// Mitsubishi GX Works2 project: VentiladoresV5   PLC: FX3G
// VentiladoresAndreDC

// global labels: Global1
VAR_GLOBAL
  Frecuencia_Actual_Cocina_Boilers AT D100 : INT;
  Corriente_Actual_Cocina_Boilers AT D102 : INT;
  Alarma_Cocina_Boilers AT M0 : BOOL;
  Automatico_Cocina_Boilers AT M1 : BOOL;
  Encender_Manual_Cocina_Boilers AT M2 : BOOL;
  Apagar_Manual_Cocina_Boilers AT M3 : BOOL;
  Reset_Alarma_Cocina_Boilers AT M4 : BOOL;
  Hora_Encendido_Cocina_Boilers AT D104 : INT;
  Minuto_Encendido_Cocina_Boilers AT D106 : INT;
  Hora_Apagado_Cocina_Boilers AT D108 : INT;
  Minuto_Apagado_Cocina_Boilers AT D110 : INT;
  SP_Velocidad_Cocina_Boilers AT D112 : INT;
  Alarma_Suministro1 AT M10 : BOOL;
  Automatico_Suministro1 AT M11 : BOOL;
  Encender_Manual_Suministro1 AT M12 : BOOL;
  Apagar_Manual_Suministro1 AT M13 : BOOL;
  Reset_Alarma_Suministro1 AT M14 : BOOL;
  Frecuencia_Actual_Suministro1 AT D114 : INT;
  Corriente_Actual_Suministro1 AT D116 : INT;
  Hora_Encendido_Suministro1 AT D118 : INT;
  Minuto_Encendido_Suministro1 AT D120 : INT;
  Hora_Apagado_Suministro1 AT D122 : INT;
  Minuto_Apagado_Suministro1 AT D124 : INT;
  SP_Velocidad_Suministro1 AT D126 : INT;
  Alarma_Suministro2 AT M20 : BOOL;
  Automatico_Suministro2 AT M21 : BOOL;
  Encender_Manual_Suministro2 AT M22 : BOOL;
  Apagar_Manual_Suministro2 AT M23 : BOOL;
  Reset_Alarma_Suministro2 AT M24 : BOOL;
  Frecuencia_Actual_Suministro2 AT D128 : INT;
  Corriente_Actual_Suministro2 AT D130 : INT;
  Hora_Encendido_Suministro2 AT D132 : INT;
  Minuto_Encendido_Suministro2 AT D134 : INT;
  Hora_Apagado_Suministro2 AT D136 : INT;
  Minuto_Apagado_Suministro2 AT D138 : INT;
  SP_Velocidad_Suministro2 AT D140 : INT;
  Alarma_Cocina_Fria AT M30 : BOOL;
  Automatico_Cocina_Fria AT M31 : BOOL;
  Encender_Manual_Cocina_Fria AT M32 : BOOL;
  Apagar_Manual_Cocina_Fria AT M33 : BOOL;
  Reset_Alarma_Cocina_Fria AT M34 : BOOL;
  Frecuencia_Actual_Cocina_Fria AT D142 : INT;
  Corriente_Actual_Cocina_Fria AT D144 : INT;
  Hora_Encendido_Cocina_Fria AT D146 : INT;
  Minuto_Encendido_Cocina_Fria AT D148 : INT;
  Hora_Apagado_Cocina_Fria AT D150 : INT;
  Minuto_Apagado_Cocina_Fria AT D152 : INT;
  SP_Velocidad_Cocina_Fria AT D154 : INT;
  Alarma_Campana_Grande AT M40 : BOOL;
  Automatico_Campana_Grande AT M41 : BOOL;
  Encender_Manual_Campana_Grande AT M42 : BOOL;
  Apagar_Manual_Campana_Grande AT M43 : BOOL;
  Reset_Alarma_Campana_Grande AT M44 : BOOL;
  Frecuencia_Actual_Campana_Grande AT D156 : INT;
  Corriente_Actual_Campana_Grande AT D158 : INT;
  Hora_Encendido_Campana_Grande AT D160 : INT;
  Minuto_Encendido_Campana_Grande AT D162 : INT;
  Hora_Apagado_Campana_Grande AT D164 : INT;
  Minuto_Apagado_Campana_Grande AT D166 : INT;
  SP_Velocidad_Campana_Grande AT D168 : INT;
  Alarma_Fachada1 AT M50 : BOOL;
  Automatico_Fachada1 AT M51 : BOOL;
  Encender_Manual_Fachada1 AT M52 : BOOL;
  Apagar_Manual_Fachada1 AT M53 : BOOL;
  Reset_Alarma_Fachada1 AT M54 : BOOL;
  Frecuencia_Actual_Fachada1 AT D170 : INT;
  Corriente_Actual_Fachada1 AT D172 : INT;
  Hora_Encendido_Fachada1 AT D174 : INT;
  Minuto_Encendido_Fachada1 AT D176 : INT;
  Hora_Apagado_Fachada1 AT D178 : INT;
  Minuto_Apagado_Fachada1 AT D180 : INT;
  SP_Velocidad_Fachada1 AT D182 : INT;
  Alarma_Fachada2 AT M60 : BOOL;
  Automatico_Fachada2 AT M61 : BOOL;
  Encender_Manual_Fachada2 AT M62 : BOOL;
  Apagar_Manual_Fachada2 AT M63 : BOOL;
  Reset_Alarma_Fachada2 AT M64 : BOOL;
  Frecuencia_Actual_Fachada2 AT D184 : INT;
  Corriente_Actual_Fachada2 AT D186 : INT;
  Hora_Encendido_Fachada2 AT D188 : INT;
  Minuto_Encendido_Fachada2 AT D190 : INT;
  Hora_Apagado_Fachada2 AT D192 : INT;
  Minuto_Apagado_Fachada2 AT D194 : INT;
  SP_Velocidad_Fachada2 AT D196 : INT;
  Alarma_Cocina_Terraza AT M70 : BOOL;
  Automatico_Cocina_Terraza AT M71 : BOOL;
  Encender_Manual_Cocina_Terraza AT M72 : BOOL;
  Apagar_Manual_Cocina_Terraza AT M73 : BOOL;
  Reset_Alarma_Cocina_Terraza AT M74 : BOOL;
  Frecuencia_Actual_Cocina_Terraza AT D198 : INT;
  Corriente_Actual_Cocina_Terraza AT D200 : INT;
  Hora_Encendido_Cocina_Terraza AT D202 : INT;
  Minuto_Encendido_Cocina_Terraza AT D204 : INT;
  Hora_Apagado_Cocina_Terraza AT D206 : INT;
  Minuto_Apagado_Cocina_Terraza AT D208 : INT;
  SP_Velocidad_Cocina_Terraza AT D210 : INT;
  Cambiar_SP_Cocina_Boilers AT M5 : BOOL;
  Cambiar_SP_Suministro1 AT M15 : BOOL;
  Cambiar_SP_Suminsitro2 AT M25 : BOOL;
  Cambiar_SP_Cocina_Fria AT M35 : BOOL;
  Cambiar_SP_Campana_Grande AT M45 : BOOL;
  Cambiar_SP_Fachada1 AT M55 : BOOL;
  Cambiar_SP_Fachada2 AT M65 : BOOL;
  Cambiar_SP_Terraza AT M75 : BOOL;
  Ultima_Alarma_Cocina_Boilers AT D212 : INT;
  Ultima_Alarma_Suministro1 AT D214 : INT;
  Ultima_Alarma_Suministro2 AT D216 : INT;
  Ultima_Alarma_Cocina_Fria AT D218 : INT;
  Ultima_Alarma_Campana_Grande AT D220 : INT;
  Ultima_Alarma_Fachada1 AT D222 : INT;
  Ultima_Alarma_Fachada2 AT D224 : INT;
  Ultima_Alarma_Cocina_Terraza AT D226 : INT;
END_VAR

// task Task_01 (event TRUE, interval 0, priority 31): Inicio_Modbus, Campana_Grande, Cocina_Boilers, Cocina_Fria, Cocina_Terraza, Fachada1, Fachada2, Suministro1, Suministro2

PROGRAM Inicio_Modbus
(* structured ladder/FBD written out as ST: instructions are called as NAME(EN, inputs, outputs); _pN, _eN, _tN stand for wires *)
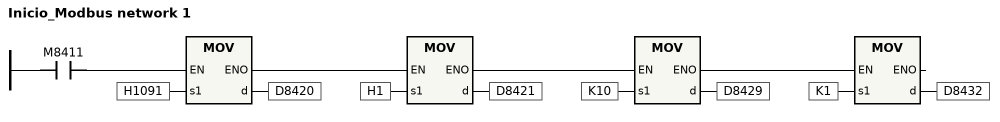
(* network 1 *)
_e1 := MOV(M8411, H1091, D8420);
_e2 := MOV(_e1, H1, D8421);
_e3 := MOV(_e2, K10, D8429);
MOV(_e3, K1, D8432);
END_PROGRAM

FUNCTION_BLOCK Comparador_Horario
VAR_INPUT
  Minuto_Encendido : INT;
  Hora_Encendido : INT;
  Minuto_Apagado : INT;
  Hora_Apagado : INT;
END_VAR
VAR
  Minuto_Encendido_Ok : BOOL;
  Hora_Encendido_Ok : BOOL;
  Minuto_Apagado_Ok : BOOL;
  Hora_Apagado_Ok : BOOL;
END_VAR
VAR_OUTPUT
  Dentro_Horario : BOOL;
END_VAR
VAR
  Encender : BOOL;
  Apagar : BOOL;
END_VAR
(* structured ladder/FBD written out as ST: instructions are called as NAME(EN, inputs, outputs); _pN, _eN, _tN stand for wires *)
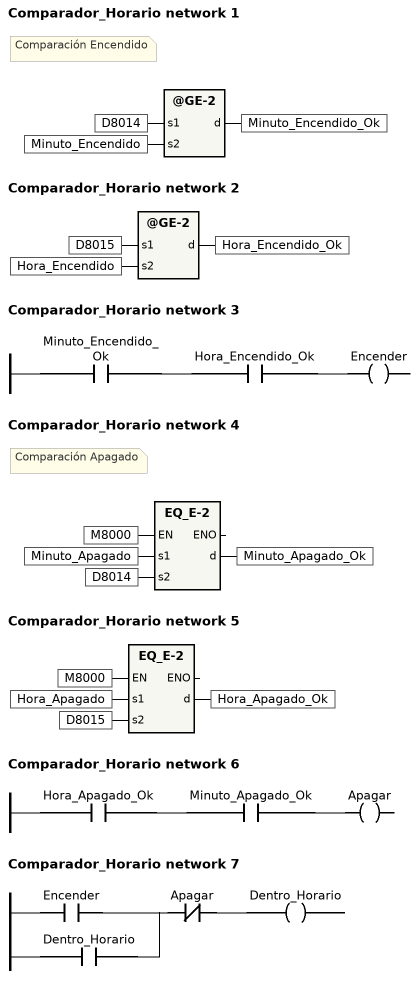
(* network 1 *)
(* Comparación Encendido *)
Minuto_Encendido_Ok := @GE-2(D8014, Minuto_Encendido);
(* network 2 *)
Hora_Encendido_Ok := @GE-2(D8015, Hora_Encendido);
(* network 3 *)
Encender := Minuto_Encendido_Ok AND Hora_Encendido_Ok;
(* network 4 *)
(* Comparación Apagado *)
EQ_E(M8000, Minuto_Apagado, D8014, Minuto_Apagado_Ok);
(* network 5 *)
EQ_E(M8000, Hora_Apagado, D8015, Hora_Apagado_Ok);
(* network 6 *)
Apagar := Hora_Apagado_Ok AND Minuto_Apagado_Ok;
(* network 7 *)
Dentro_Horario := (Encender OR Dentro_Horario) AND NOT Apagar;
END_FUNCTION_BLOCK

FUNCTION_BLOCK Control_Variador_Mitsubishi
VAR_INPUT
  Automatico : BOOL;
  Encender_Manual : BOOL;
  Hora_Encendido : INT;
  Minuto_Encendido : INT;
  SP_Velocidad : INT;
  Direccion_Modbus : INT;
END_VAR
VAR
  Comparador_Horario_1 : Comparador_Horario;
END_VAR
VAR_INPUT
  Minuto_Apagado : INT;
  Hora_Apagado : INT;
END_VAR
VAR
  Horario_Ok : BOOL;
  Encender_Variador_Automatico : BOOL;
  Apagar_Variador_Automatico : BOOL;
END_VAR
VAR_INPUT
  Apagar_Manual : BOOL;
END_VAR
VAR
  TP_1 : TP;
  TP_2 : TP;
END_VAR
VAR_INPUT
  Reset_Alarma : BOOL;
  Cambiar_SP : BOOL;
END_VAR
(* structured ladder/FBD written out as ST: instructions are called as NAME(EN, inputs, outputs); _pN, _eN, _tN stand for wires *)
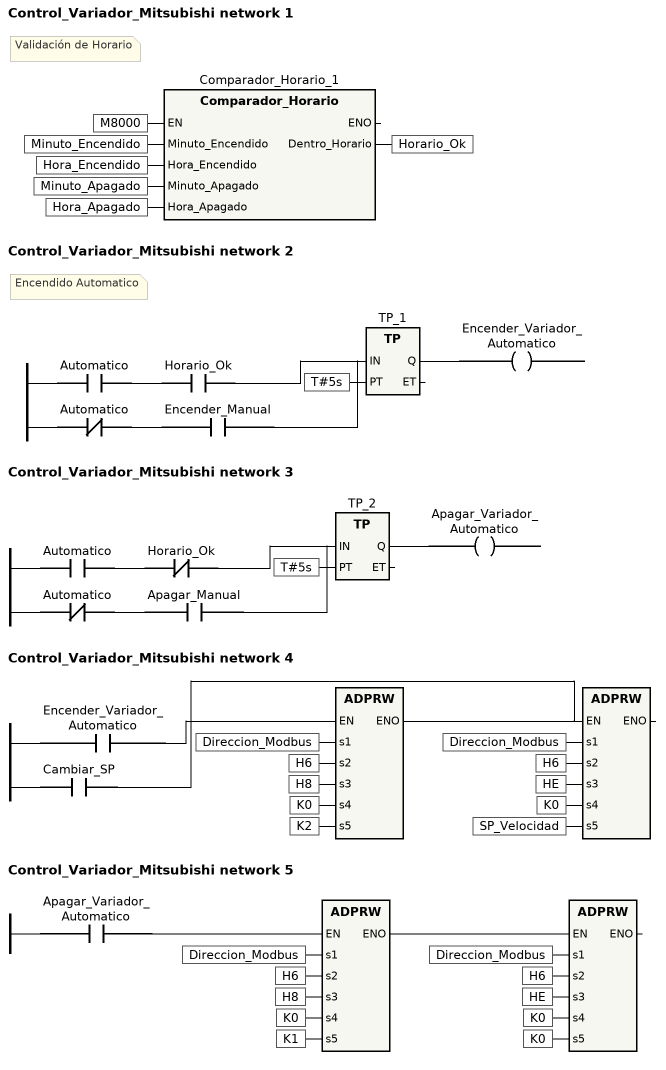
(* network 1 *)
(* Validación de Horario *)
Comparador_Horario_1(EN := M8000, Minuto_Encendido := Minuto_Encendido, Hora_Encendido := Hora_Encendido, Minuto_Apagado := Minuto_Apagado, Hora_Apagado := Hora_Apagado, Dentro_Horario => Horario_Ok);
(* network 2 *)
(* Encendido Automatico *)
TP_1(IN := (Automatico AND Horario_Ok) OR (NOT Automatico AND Encender_Manual), PT := T#5s);
Encender_Variador_Automatico := TP_1.Q;
(* network 3 *)
TP_2(IN := (Automatico AND NOT Horario_Ok) OR (NOT Automatico AND Apagar_Manual), PT := T#5s);
Apagar_Variador_Automatico := TP_2.Q;
(* network 4 *)
_e1 := ADPRW(Encender_Variador_Automatico, Direccion_Modbus, H6, H8, K0, K2);
ADPRW(_e1 OR Cambiar_SP, Direccion_Modbus, H6, HE, K0, SP_Velocidad);
(* network 5 *)
_e1 := ADPRW(Apagar_Variador_Automatico, Direccion_Modbus, H6, H8, K0, K1);
ADPRW(_e1, Direccion_Modbus, H6, HE, K0, K0);
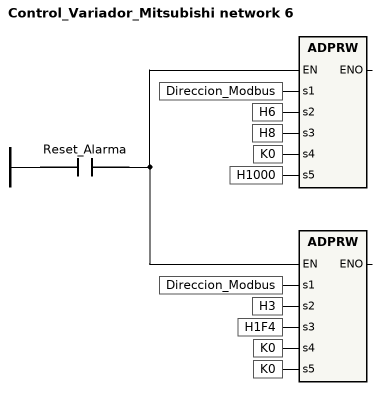
(* network 6 *)
ADPRW(Reset_Alarma, Direccion_Modbus, H6, H8, K0, H1000);
ADPRW(Reset_Alarma, Direccion_Modbus, H3, H1F4, K0, K0);
END_FUNCTION_BLOCK

FUNCTION_BLOCK Lectura_Variador_Mitsubishi
VAR_INPUT
  Direccion_Modbus : INT;
END_VAR
VAR_OUTPUT
  Frecuencia_Actual : INT;
  Corriente_Actual : INT;
  Alarma : BOOL;
END_VAR
VAR
  Estado_VFD : INT;
END_VAR
VAR_OUTPUT
  Ultima_Alarma : INT;
END_VAR
(* structured ladder/FBD written out as ST: instructions are called as NAME(EN, inputs, outputs); _pN, _eN, _tN stand for wires *)
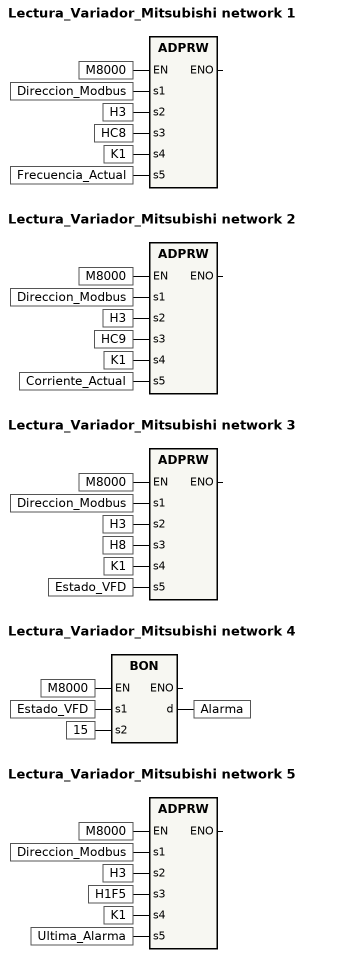
(* network 1 *)
ADPRW(M8000, Direccion_Modbus, H3, HC8, K1, Frecuencia_Actual);
(* network 2 *)
ADPRW(M8000, Direccion_Modbus, H3, HC9, K1, Corriente_Actual);
(* network 3 *)
ADPRW(M8000, Direccion_Modbus, H3, H8, K1, Estado_VFD);
(* network 4 *)
BON(M8000, Estado_VFD, 15, Alarma);
(* network 5 *)
ADPRW(M8000, Direccion_Modbus, H3, H1F5, K1, Ultima_Alarma);
END_FUNCTION_BLOCK

PROGRAM Cocina_Boilers
VAR
  Lectura_Variador_Mitsubishi_1 : Lectura_Variador_Mitsubishi;
  Control_Variador_Mitsubishi_1 : Control_Variador_Mitsubishi;
END_VAR
(* structured ladder/FBD written out as ST: instructions are called as NAME(EN, inputs, outputs); _pN, _eN, _tN stand for wires *)
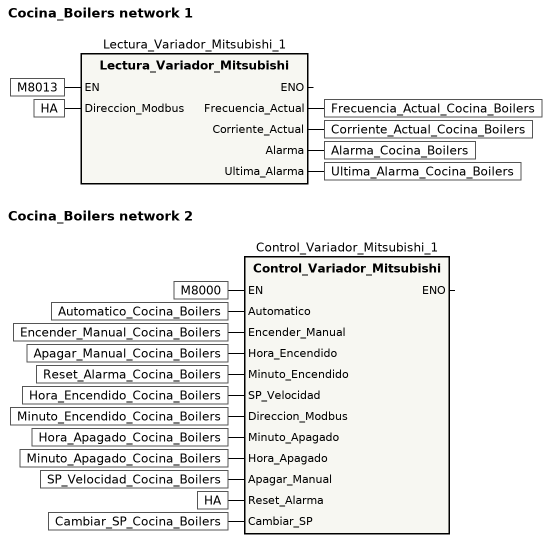
(* network 1 *)
Lectura_Variador_Mitsubishi_1(EN := M8013, Direccion_Modbus := HA, Frecuencia_Actual => Frecuencia_Actual_Cocina_Boilers, Corriente_Actual => Corriente_Actual_Cocina_Boilers, Alarma => Alarma_Cocina_Boilers, Ultima_Alarma => Ultima_Alarma_Cocina_Boilers);
(* network 2 *)
Control_Variador_Mitsubishi_1(EN := M8000, Automatico := Automatico_Cocina_Boilers, Encender_Manual := Encender_Manual_Cocina_Boilers, Hora_Encendido := Apagar_Manual_Cocina_Boilers, Minuto_Encendido := Reset_Alarma_Cocina_Boilers, SP_Velocidad := Hora_Encendido_Cocina_Boilers, Direccion_Modbus := Minuto_Encendido_Cocina_Boilers, Minuto_Apagado := Hora_Apagado_Cocina_Boilers, Hora_Apagado := Minuto_Apagado_Cocina_Boilers, Apagar_Manual := SP_Velocidad_Cocina_Boilers, Reset_Alarma := HA, Cambiar_SP := Cambiar_SP_Cocina_Boilers);
END_PROGRAM

FUNCTION_BLOCK Control_Variador_Altivar
VAR_INPUT
  Automatico : BOOL;
  Encender_Manual : BOOL;
  Hora_Encendido : INT;
  Minuto_Encendido : INT;
  SP_Velocidad : INT;
  Direccion_Modbus : INT;
END_VAR
VAR
  Comparador_Horario_1 : Comparador_Horario;
END_VAR
VAR_INPUT
  Minuto_Apagado : INT;
  Hora_Apagado : INT;
END_VAR
VAR
  Horario_Ok : BOOL;
  Encender_Variador_Automatico : BOOL;
  Apagar_Variador_Automatico : BOOL;
END_VAR
VAR_INPUT
  Apagar_Manual : BOOL;
END_VAR
VAR
  TP_1 : TP;
  TP_2 : TP;
END_VAR
VAR_INPUT
  Reset_Alarma : BOOL;
  Cambiar_SP : BOOL;
END_VAR
(* structured ladder/FBD written out as ST: instructions are called as NAME(EN, inputs, outputs); _pN, _eN, _tN stand for wires *)
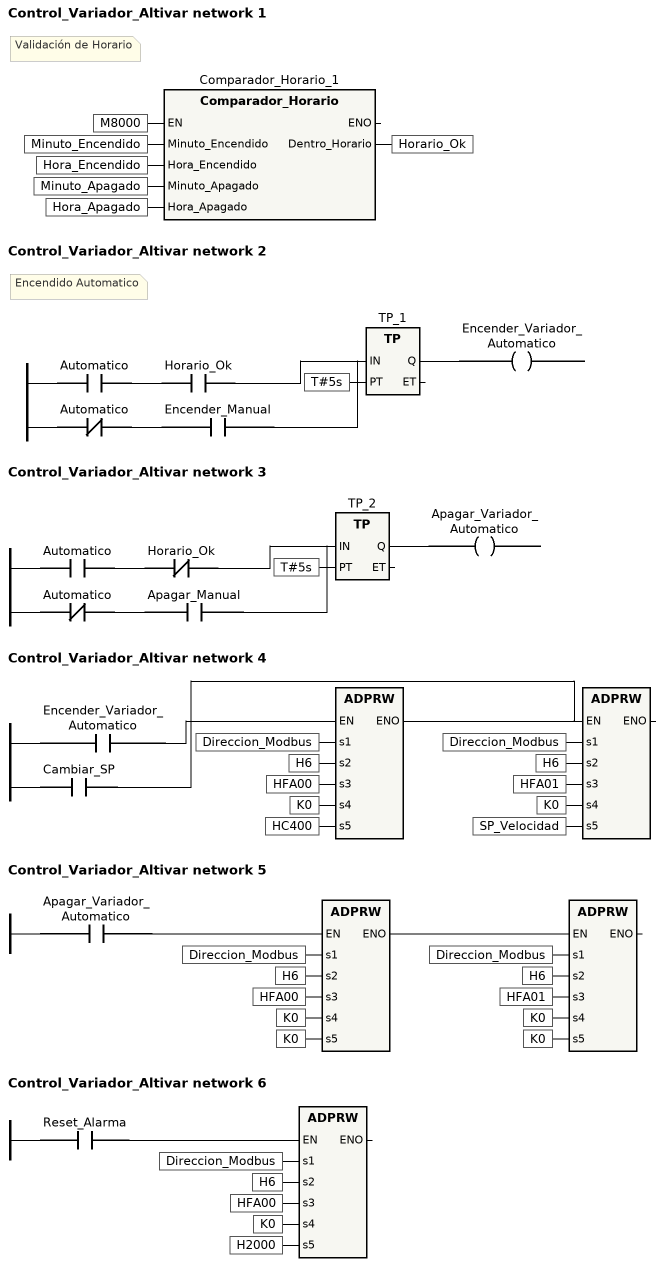
(* network 1 *)
(* Validación de Horario *)
Comparador_Horario_1(EN := M8000, Minuto_Encendido := Minuto_Encendido, Hora_Encendido := Hora_Encendido, Minuto_Apagado := Minuto_Apagado, Hora_Apagado := Hora_Apagado, Dentro_Horario => Horario_Ok);
(* network 2 *)
(* Encendido Automatico *)
TP_1(IN := (Automatico AND Horario_Ok) OR (NOT Automatico AND Encender_Manual), PT := T#5s);
Encender_Variador_Automatico := TP_1.Q;
(* network 3 *)
TP_2(IN := (Automatico AND NOT Horario_Ok) OR (NOT Automatico AND Apagar_Manual), PT := T#5s);
Apagar_Variador_Automatico := TP_2.Q;
(* network 4 *)
_e1 := ADPRW(Encender_Variador_Automatico, Direccion_Modbus, H6, HFA00, K0, HC400);
ADPRW(_e1 OR Cambiar_SP, Direccion_Modbus, H6, HFA01, K0, SP_Velocidad);
(* network 5 *)
_e1 := ADPRW(Apagar_Variador_Automatico, Direccion_Modbus, H6, HFA00, K0, K0);
ADPRW(_e1, Direccion_Modbus, H6, HFA01, K0, K0);
(* network 6 *)
ADPRW(Reset_Alarma, Direccion_Modbus, H6, HFA00, K0, H2000);
END_FUNCTION_BLOCK

FUNCTION_BLOCK Lectura_Variador_Altivar
VAR_INPUT
  Direccion_Modbus : INT;
END_VAR
VAR_OUTPUT
  Frecuencia_Actual : INT;
  Corriente_Actual : INT;
  Alarma : BOOL;
END_VAR
VAR
  Estado_VFD : INT;
END_VAR
VAR_OUTPUT
  Ultima_Alarma : INT;
END_VAR
(* structured ladder/FBD written out as ST: instructions are called as NAME(EN, inputs, outputs); _pN, _eN, _tN stand for wires *)
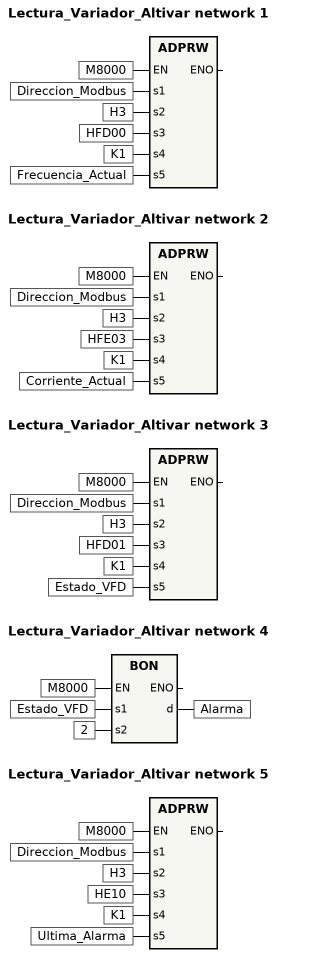
(* network 1 *)
ADPRW(M8000, Direccion_Modbus, H3, HFD00, K1, Frecuencia_Actual);
(* network 2 *)
ADPRW(M8000, Direccion_Modbus, H3, HFE03, K1, Corriente_Actual);
(* network 3 *)
ADPRW(M8000, Direccion_Modbus, H3, HFD01, K1, Estado_VFD);
(* network 4 *)
BON(M8000, Estado_VFD, 2, Alarma);
(* network 5 *)
ADPRW(M8000, Direccion_Modbus, H3, HE10, K1, Ultima_Alarma);
END_FUNCTION_BLOCK

PROGRAM Cocina_Terraza
VAR
  Lectura_Variador_Altivar_1 : Lectura_Variador_Altivar;
  Control_Variador_Altivar_1 : Control_Variador_Altivar;
END_VAR
(* structured ladder/FBD written out as ST: instructions are called as NAME(EN, inputs, outputs); _pN, _eN, _tN stand for wires *)
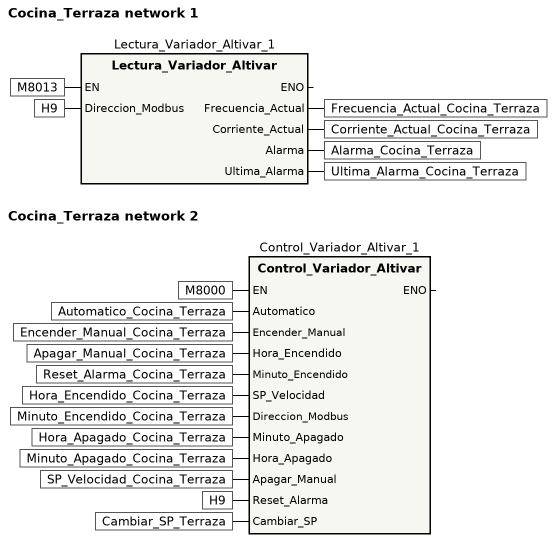
(* network 1 *)
Lectura_Variador_Altivar_1(EN := M8013, Direccion_Modbus := H9, Frecuencia_Actual => Frecuencia_Actual_Cocina_Terraza, Corriente_Actual => Corriente_Actual_Cocina_Terraza, Alarma => Alarma_Cocina_Terraza, Ultima_Alarma => Ultima_Alarma_Cocina_Terraza);
(* network 2 *)
Control_Variador_Altivar_1(EN := M8000, Automatico := Automatico_Cocina_Terraza, Encender_Manual := Encender_Manual_Cocina_Terraza, Hora_Encendido := Apagar_Manual_Cocina_Terraza, Minuto_Encendido := Reset_Alarma_Cocina_Terraza, SP_Velocidad := Hora_Encendido_Cocina_Terraza, Direccion_Modbus := Minuto_Encendido_Cocina_Terraza, Minuto_Apagado := Hora_Apagado_Cocina_Terraza, Hora_Apagado := Minuto_Apagado_Cocina_Terraza, Apagar_Manual := SP_Velocidad_Cocina_Terraza, Reset_Alarma := H9, Cambiar_SP := Cambiar_SP_Terraza);
END_PROGRAM

PROGRAM Suministro1
VAR
  Lectura_Variador_Mitsubishi_1 : Lectura_Variador_Mitsubishi;
  Control_Variador_Mitsubishi_1 : Control_Variador_Mitsubishi;
END_VAR
(* structured ladder/FBD written out as ST: instructions are called as NAME(EN, inputs, outputs); _pN, _eN, _tN stand for wires *)
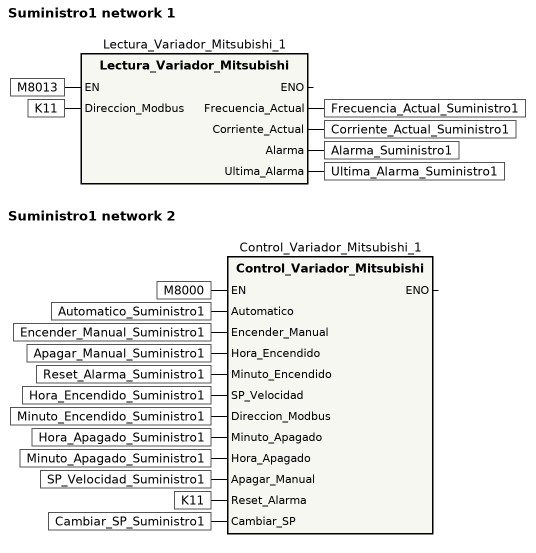
(* network 1 *)
Lectura_Variador_Mitsubishi_1(EN := M8013, Direccion_Modbus := K11, Frecuencia_Actual => Frecuencia_Actual_Suministro1, Corriente_Actual => Corriente_Actual_Suministro1, Alarma => Alarma_Suministro1, Ultima_Alarma => Ultima_Alarma_Suministro1);
(* network 2 *)
Control_Variador_Mitsubishi_1(EN := M8000, Automatico := Automatico_Suministro1, Encender_Manual := Encender_Manual_Suministro1, Hora_Encendido := Apagar_Manual_Suministro1, Minuto_Encendido := Reset_Alarma_Suministro1, SP_Velocidad := Hora_Encendido_Suministro1, Direccion_Modbus := Minuto_Encendido_Suministro1, Minuto_Apagado := Hora_Apagado_Suministro1, Hora_Apagado := Minuto_Apagado_Suministro1, Apagar_Manual := SP_Velocidad_Suministro1, Reset_Alarma := K11, Cambiar_SP := Cambiar_SP_Suministro1);
END_PROGRAM

PROGRAM Suministro2
VAR
  Lectura_Variador_Altivar_1 : Lectura_Variador_Altivar;
  Control_Variador_Altivar_1 : Control_Variador_Altivar;
END_VAR
(* structured ladder/FBD written out as ST: instructions are called as NAME(EN, inputs, outputs); _pN, _eN, _tN stand for wires *)
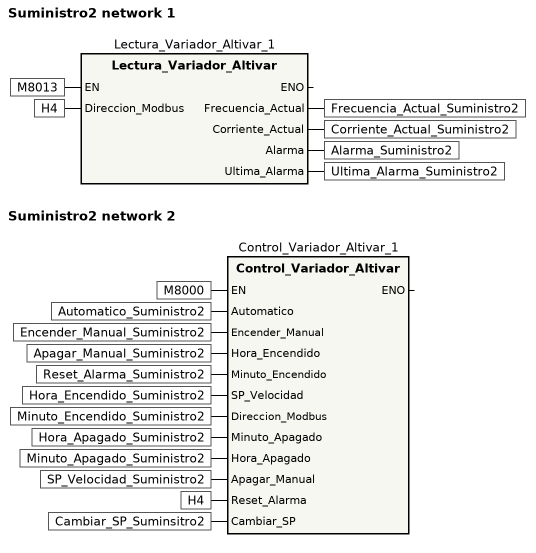
(* network 1 *)
Lectura_Variador_Altivar_1(EN := M8013, Direccion_Modbus := H4, Frecuencia_Actual => Frecuencia_Actual_Suministro2, Corriente_Actual => Corriente_Actual_Suministro2, Alarma => Alarma_Suministro2, Ultima_Alarma => Ultima_Alarma_Suministro2);
(* network 2 *)
Control_Variador_Altivar_1(EN := M8000, Automatico := Automatico_Suministro2, Encender_Manual := Encender_Manual_Suministro2, Hora_Encendido := Apagar_Manual_Suministro2, Minuto_Encendido := Reset_Alarma_Suministro2, SP_Velocidad := Hora_Encendido_Suministro2, Direccion_Modbus := Minuto_Encendido_Suministro2, Minuto_Apagado := Hora_Apagado_Suministro2, Hora_Apagado := Minuto_Apagado_Suministro2, Apagar_Manual := SP_Velocidad_Suministro2, Reset_Alarma := H4, Cambiar_SP := Cambiar_SP_Suminsitro2);
END_PROGRAM

PROGRAM Fachada1
VAR
  Lectura_Variador_Altivar_1 : Lectura_Variador_Altivar;
  Control_Variador_Altivar_1 : Control_Variador_Altivar;
END_VAR
(* structured ladder/FBD written out as ST: instructions are called as NAME(EN, inputs, outputs); _pN, _eN, _tN stand for wires *)
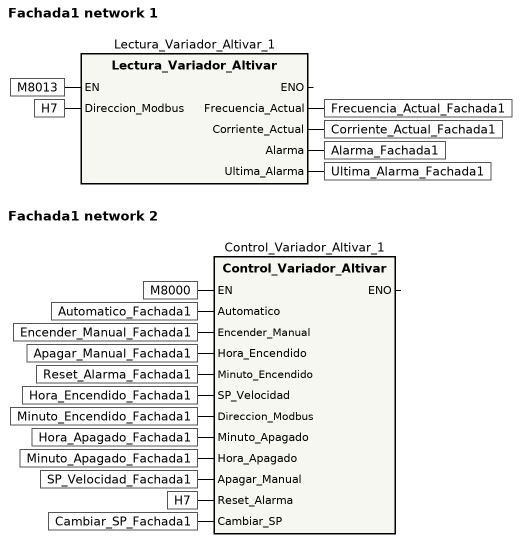
(* network 1 *)
Lectura_Variador_Altivar_1(EN := M8013, Direccion_Modbus := H7, Frecuencia_Actual => Frecuencia_Actual_Fachada1, Corriente_Actual => Corriente_Actual_Fachada1, Alarma => Alarma_Fachada1, Ultima_Alarma => Ultima_Alarma_Fachada1);
(* network 2 *)
Control_Variador_Altivar_1(EN := M8000, Automatico := Automatico_Fachada1, Encender_Manual := Encender_Manual_Fachada1, Hora_Encendido := Apagar_Manual_Fachada1, Minuto_Encendido := Reset_Alarma_Fachada1, SP_Velocidad := Hora_Encendido_Fachada1, Direccion_Modbus := Minuto_Encendido_Fachada1, Minuto_Apagado := Hora_Apagado_Fachada1, Hora_Apagado := Minuto_Apagado_Fachada1, Apagar_Manual := SP_Velocidad_Fachada1, Reset_Alarma := H7, Cambiar_SP := Cambiar_SP_Fachada1);
END_PROGRAM

PROGRAM Fachada2
VAR
  Lectura_Variador_Altivar_1 : Lectura_Variador_Altivar;
  Control_Variador_Altivar_1 : Control_Variador_Altivar;
END_VAR
(* structured ladder/FBD written out as ST: instructions are called as NAME(EN, inputs, outputs); _pN, _eN, _tN stand for wires *)
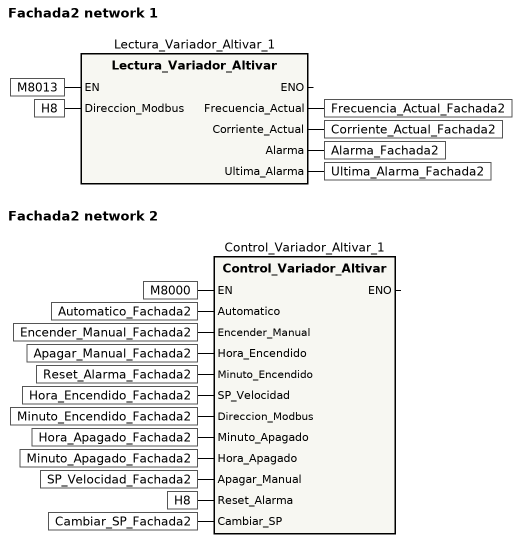
(* network 1 *)
Lectura_Variador_Altivar_1(EN := M8013, Direccion_Modbus := H8, Frecuencia_Actual => Frecuencia_Actual_Fachada2, Corriente_Actual => Corriente_Actual_Fachada2, Alarma => Alarma_Fachada2, Ultima_Alarma => Ultima_Alarma_Fachada2);
(* network 2 *)
Control_Variador_Altivar_1(EN := M8000, Automatico := Automatico_Fachada2, Encender_Manual := Encender_Manual_Fachada2, Hora_Encendido := Apagar_Manual_Fachada2, Minuto_Encendido := Reset_Alarma_Fachada2, SP_Velocidad := Hora_Encendido_Fachada2, Direccion_Modbus := Minuto_Encendido_Fachada2, Minuto_Apagado := Hora_Apagado_Fachada2, Hora_Apagado := Minuto_Apagado_Fachada2, Apagar_Manual := SP_Velocidad_Fachada2, Reset_Alarma := H8, Cambiar_SP := Cambiar_SP_Fachada2);
END_PROGRAM

PROGRAM Campana_Grande
VAR
  Lectura_Variador_Altivar_1 : Lectura_Variador_Altivar;
  Control_Variador_Altivar_1 : Control_Variador_Altivar;
END_VAR
(* structured ladder/FBD written out as ST: instructions are called as NAME(EN, inputs, outputs); _pN, _eN, _tN stand for wires *)
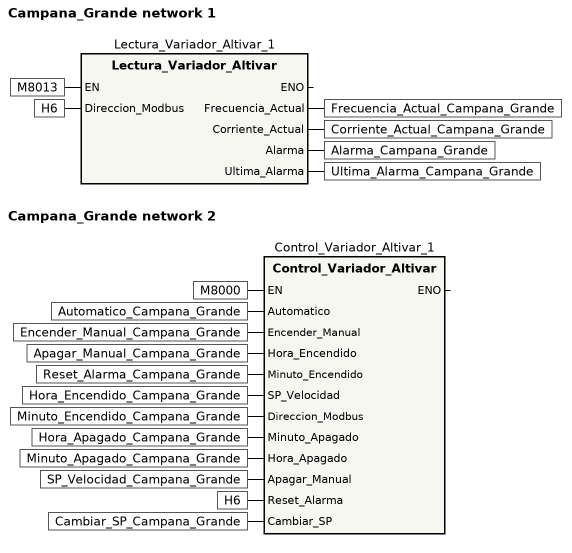
(* network 1 *)
Lectura_Variador_Altivar_1(EN := M8013, Direccion_Modbus := H6, Frecuencia_Actual => Frecuencia_Actual_Campana_Grande, Corriente_Actual => Corriente_Actual_Campana_Grande, Alarma => Alarma_Campana_Grande, Ultima_Alarma => Ultima_Alarma_Campana_Grande);
(* network 2 *)
Control_Variador_Altivar_1(EN := M8000, Automatico := Automatico_Campana_Grande, Encender_Manual := Encender_Manual_Campana_Grande, Hora_Encendido := Apagar_Manual_Campana_Grande, Minuto_Encendido := Reset_Alarma_Campana_Grande, SP_Velocidad := Hora_Encendido_Campana_Grande, Direccion_Modbus := Minuto_Encendido_Campana_Grande, Minuto_Apagado := Hora_Apagado_Campana_Grande, Hora_Apagado := Minuto_Apagado_Campana_Grande, Apagar_Manual := SP_Velocidad_Campana_Grande, Reset_Alarma := H6, Cambiar_SP := Cambiar_SP_Campana_Grande);
END_PROGRAM

PROGRAM Cocina_Fria
VAR
  Lectura_Variador_Altivar_1 : Lectura_Variador_Altivar;
  Control_Variador_Altivar_1 : Control_Variador_Altivar;
END_VAR
(* structured ladder/FBD written out as ST: instructions are called as NAME(EN, inputs, outputs); _pN, _eN, _tN stand for wires *)
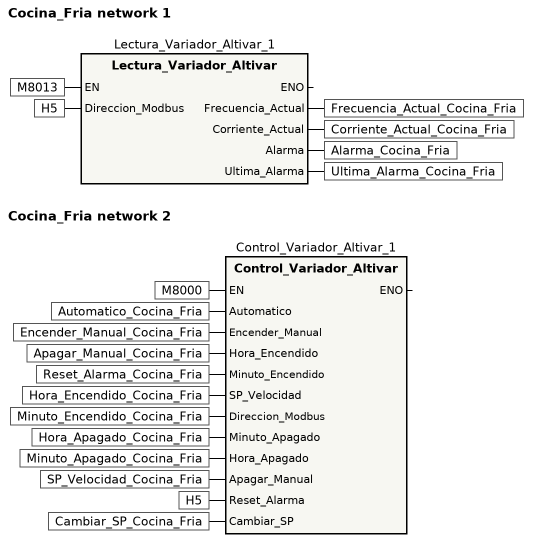
(* network 1 *)
Lectura_Variador_Altivar_1(EN := M8013, Direccion_Modbus := H5, Frecuencia_Actual => Frecuencia_Actual_Cocina_Fria, Corriente_Actual => Corriente_Actual_Cocina_Fria, Alarma => Alarma_Cocina_Fria, Ultima_Alarma => Ultima_Alarma_Cocina_Fria);
(* network 2 *)
Control_Variador_Altivar_1(EN := M8000, Automatico := Automatico_Cocina_Fria, Encender_Manual := Encender_Manual_Cocina_Fria, Hora_Encendido := Apagar_Manual_Cocina_Fria, Minuto_Encendido := Reset_Alarma_Cocina_Fria, SP_Velocidad := Hora_Encendido_Cocina_Fria, Direccion_Modbus := Minuto_Encendido_Cocina_Fria, Minuto_Apagado := Hora_Apagado_Cocina_Fria, Hora_Apagado := Minuto_Apagado_Cocina_Fria, Apagar_Manual := SP_Velocidad_Cocina_Fria, Reset_Alarma := H5, Cambiar_SP := Cambiar_SP_Cocina_Fria);
END_PROGRAM
